{attribute 'GeneratedUsingTerminal: EL6002-0000-0019'}
{attribute addProperty BoxType "EL6002-0000-0019"}
{attribute addProperty Id "StatusAT %I*UINT2Data_InAT %I*ARRAY[0..21] OF USINT22"}
{attribute addProperty CRC "1367962124"}
{attribute addProperty Size "24"}
TYPE COM_TxPDO_Map_Inputs_Channel_6C2FC202 EXTENDS InputBase_8311D824 :
STRUCT
	{attribute addProperty Name "Status"}
	Status AT %I* : UINT;
	{attribute addProperty Name "Data_In"}
	Data_In AT %I* : ARRAY[0..21] OF USINT;
END_STRUCT
END_TYPE

(* stored: Version 1.2.0.0, ProductVersion 3.1.4024.11
   DUT COM_TxPDO_Map_Inputs_Channel_6C2FC202: Id {da232a6a-7260-4a8c-b029-d72b7543f842} *)
